FUNCTION "Array_Int.Shift_Down" : Void
{ S7_Optimized_Access := 'TRUE' }
VERSION : 0.1
   VAR_INPUT
      null_token : Int;
   END_VAR

   VAR_IN_OUT
      source_arrary : Variant;
   END_VAR

   VAR_TEMP
      i : Int;
      _array : Array[0..999] of Int;
      len_array : UDInt;
      status : Int;
      ubound : Int;
   END_VAR


BEGIN
	REGION "GET LENGTH"
	    #len_array := CountOfElements(#source_arrary);
	END_REGION

	REGION "COPY TO LOCAL"
	    #status := MOVE_BLK_VARIANT(SRC := #source_arrary,
	                                COUNT := #len_array,
	                                SRC_INDEX := 0,
	                                DEST_INDEX := 0,
	                                DEST => #_array);
	END_REGION


	REGION "FILL LENGTH WITH BYTE IN"
	    #ubound := UDINT_TO_INT(#len_array) - 1;
	    FOR #i := 0 TO #ubound DO
	        IF #i = #ubound THEN
	            #_array[#i] := #null_token;
	            CONTINUE;
	        END_IF;
	        #_array[#i] := #_array[#i + 1];
	    END_FOR;
	END_REGION


	REGION "RETURN"
	    #status := MOVE_BLK_VARIANT(SRC := #_array,
	                                COUNT := #len_array,
	                                SRC_INDEX := 0,
	                                DEST_INDEX := 0,
	                                DEST => #source_arrary);
	END_REGION

END_FUNCTION

